{attribute 'enable_dynamic_creation'}
FUNCTION_BLOCK FB_Rectangle IMPLEMENTS I_Shape
VAR_INPUT
END_VAR
VAR_OUTPUT
END_VAR
VAR
END_VAR

{warning 'Agregar implementación de método'}
METHOD M_Draw : BOOL
ADSLOGSTR(ADSLOG_MSGTYPE_HINT, 'Draw rectangle', '');
M_Draw := TRUE;
END_METHOD

END_FUNCTION_BLOCK

(* stored: Version 1.1.0.1, ProductVersion 3.1.4024.12
   POU FB_Rectangle: Id {1aa9c012-67ef-4b4c-9e92-2881ac0a0e05}, SpecialFunc None
   Method M_Draw: Id {52084d2b-6c2e-49dc-b2f7-ab6e76a50e30} *)
